(* IEC 61131-3 sources: POMIRTS_lab3/AS/Library_2/AsNxDpM, 3 files *)

(* ---- AsNxDpM.typ ---- *)
TYPE
	nxdpmLifeList_t			: STRUCT			(*life list*)
		node				: ARRAY[0..127] OF USINT;
	END_STRUCT;

	nxdpmDiagData_t			: STRUCT			(*diagnoctic data*)
		status1				: USINT;			(*status1*)
		status2				: USINT;			(*status2*)
		status3				: USINT;			(*status3*)
		address				: USINT;			(*address*)
		identHigh			: USINT;			(*ident high*)
		identLow			: USINT;			(*ident low*)
		blockData			: ARRAY[0..237] OF USINT;
	END_STRUCT;

	nxdpmAddAdrParam_t		: STRUCT			(*additional address parameter*)
		srcType				: USINT;
		srcSize				: USINT;
		destType			: USINT;
		destSize			: USINT;
		addParam			: ARRAY[0..227] OF USINT;
	END_STRUCT;
END_TYPE

(* ---- AsNxDpM.fun ---- *)
{REDUND_CONTEXT} {REDUND_UNREPLICABLE} FUNCTION_BLOCK nxdpmCommand				(*send command*)
	VAR_INPUT
		enable			: BOOL;			(*enables execution*)
		pDevice			: UDINT;		(*interface name given as a pointer, e.g., "SL<x>.SS<y>.IF<z>"*)
		remoteAdr		: UDINT;		(*remote address*)
		syncCommand		: UDINT;		(*sync command*)
		freezeCommand	: UDINT;		(*freeze command*)
		group			: UDINT;		(*group*)
	END_VAR
	VAR
        _state			: UINT;			(*internal variable*)
		_result			: UINT;			(*internal variable*)
        _srcId			: UDINT;		(*internal variable*)
	END_VAR
	VAR_OUTPUT
		status			: UINT;			(*execution status: ERR_OK, ERR_FUB_ENABLE_FALSE, ERR_FUB_BUSY, 0xXXXX = see help*)
		dpStatus		: UDINT;		(*profibus DP stack status*)
	END_VAR
END_FUNCTION_BLOCK

{REDUND_CONTEXT} {REDUND_UNREPLICABLE} FUNCTION_BLOCK nxdpmSetMode				(*set mode*)
	VAR_INPUT
		enable			: BOOL;			(*enables execution*)
		pDevice			: UDINT;		(*interface name given as a pointer, e.g., "SL<x>.SS<y>.IF<z>"*)
		mode			: UDINT;		(*mode to set*)
	END_VAR
	VAR
        _state			: UINT;			(*internal variable*)
		_result			: UINT;			(*internal variable*)
        _srcId			: UDINT;		(*internal variable*)
	END_VAR
	VAR_OUTPUT
		status			: UINT;			(*execution status: ERR_OK, ERR_FUB_ENABLE_FALSE, ERR_FUB_BUSY, 0xXXXX = see help*)
		dpStatus		: UDINT;		(*profibus DP stack status*)
	END_VAR
END_FUNCTION_BLOCK

{REDUND_CONTEXT} {REDUND_UNREPLICABLE} FUNCTION_BLOCK nxdpmActivate			(*activate/deactivate slave*)
	VAR_INPUT
		enable			: BOOL;			(*enables execution*)
		pDevice			: UDINT;		(*interface name given as a pointer, e.g., "SL<x>.SS<y>.IF<z>"*)
		remoteAdr		: UDINT;		(*remote address*)
		activate		: UDINT;		(*activate/deactivate slave*)
	END_VAR
	VAR
        _state			: UINT;			(*internal variable*)
		_result			: UINT;			(*internal variable*)
        _srcId			: UDINT;		(*internal variable*)
	END_VAR
	VAR_OUTPUT
		status			: UINT;			(*execution status: ERR_OK, ERR_FUB_ENABLE_FALSE, ERR_FUB_BUSY, 0xXXXX = see help*)
		dpStatus		: UDINT;		(*profibus DP stack status*)
	END_VAR
END_FUNCTION_BLOCK

{REDUND_CONTEXT} {REDUND_UNREPLICABLE} FUNCTION_BLOCK nxdpmGetDiag				(*get diagnostic*)
	VAR_INPUT
		enable			: BOOL;			(*enables execution*)
		pDevice			: UDINT;		(*interface name given as a pointer, e.g., "SL<x>.SS<y>.IF<z>"*)
		remoteAdr		: UDINT;		(*remote address*)
		flags			: UDINT;		(*flags*)
		pDiagData		: UDINT;		(*diagnostic data given as a pointer*)
	END_VAR
	VAR
        _state			: UINT;			(*internal variable*)
		_result			: UINT;			(*internal variable*)
        _srcId			: UDINT;		(*internal variable*)
	END_VAR
	VAR_OUTPUT
		status			: UINT;			(*execution status: ERR_OK, ERR_FUB_ENABLE_FALSE, ERR_FUB_BUSY, 0xXXXX = see help*)
		dpStatus		: UDINT;		(*profibus DP stack status*)
		diagDataLen		: UDINT;		(*diagnostic data length*)
	END_VAR
END_FUNCTION_BLOCK

{REDUND_CONTEXT} {REDUND_UNREPLICABLE} FUNCTION_BLOCK nxdpmLifeList			(*life list*)
	VAR_INPUT
		enable			: BOOL;			(*enables execution*)
		pDevice			: UDINT;		(*interface name given as a pointer, e.g., "SL<x>.SS<y>.IF<z>"*)
		pLifeList		: UDINT;		(*life list area given as a pointer*)
	END_VAR
	VAR
        _state			: UINT;			(*internal variable*)
		_result			: UINT;			(*internal variable*)
        _srcId			: UDINT;		(*internal variable*)
	END_VAR
	VAR_OUTPUT
		status			: UINT;			(*execution status: ERR_OK, ERR_FUB_ENABLE_FALSE, ERR_FUB_BUSY, 0xXXXX = see help*)
		dpStatus		: UDINT;		(*profibus DP stack status*)
	END_VAR
END_FUNCTION_BLOCK

{REDUND_CONTEXT} {REDUND_UNREPLICABLE} FUNCTION_BLOCK nxdpmV1C1Read			(*DPV1 class 1 read request*)
	VAR_INPUT
		enable			: BOOL;			(*enables execution*)
		pDevice			: UDINT;		(*interface name given as a pointer, e.g., "SL<x>.SS<y>.IF<z>"*)
		remoteAdr		: UDINT;		(*remote address*)
		slotNumber		: UDINT;		(*slot number*)
		index			: UDINT;		(*index*)
		dataLen			: UDINT;		(*data length*)
		pData			: UDINT;		(*data area given as a pointer*)
	END_VAR
	VAR
        _state			: UINT;			(*internal variable*)
		_result			: UINT;			(*internal variable*)
        _srcId			: UDINT;		(*internal variable*)
	END_VAR
	VAR_OUTPUT
		status			: UINT;			(*execution status: ERR_OK, ERR_FUB_ENABLE_FALSE, ERR_FUB_BUSY, 0xXXXX = see help*)
		dpStatus		: UDINT;		(*profibus DP stack status*)
		readDataLen		: UDINT;		(*read data length*)
	END_VAR
END_FUNCTION_BLOCK

{REDUND_CONTEXT} {REDUND_UNREPLICABLE} FUNCTION_BLOCK nxdpmV1C1Write			(*DPV1 class 1 write request*)
	VAR_INPUT
		enable			: BOOL;			(*enables execution*)
		pDevice			: UDINT;		(*interface name given as a pointer, e.g., "SL<x>.SS<y>.IF<z>"*)
		remoteAdr		: UDINT;		(*remote address*)
		slotNumber		: UDINT;		(*slot number*)
		index			: UDINT;		(*index*)
		dataLen			: UDINT;		(*data length*)
		pData			: UDINT;		(*data area given as a pointer*)
	END_VAR
	VAR
        _state			: UINT;			(*internal variable*)
		_result			: UINT;			(*internal variable*)
        _srcId			: UDINT;		(*internal variable*)
	END_VAR
	VAR_OUTPUT
		status			: UINT;			(*execution status: ERR_OK, ERR_FUB_ENABLE_FALSE, ERR_FUB_BUSY, 0xXXXX = see help*)
		dpStatus		: UDINT;		(*profibus DP stack status*)
		errorDecode		: USINT;		(*error decode*)
		errorCode1		: USINT;		(*error code 1*)
		errorCode2		: USINT;		(*error code 2*)
	END_VAR
END_FUNCTION_BLOCK

{REDUND_CONTEXT} {REDUND_UNREPLICABLE} FUNCTION_BLOCK nxdpmSubscribe			(*subscribe master*)
	VAR_INPUT
		enable			: BOOL;			(*enables execution*)
		pDevice			: UDINT;		(*interface name given as a pointer, e.g., "SL<x>.SS<y>.IF<z>"*)
	END_VAR
	VAR
        _state			: UINT;			(*internal variable*)
		_result			: UINT;			(*internal variable*)
        _srcId			: UDINT;		(*internal variable*)
	END_VAR
	VAR_OUTPUT
		status			: UINT;			(*execution status: ERR_OK, ERR_FUB_ENABLE_FALSE, ERR_FUB_BUSY, 0xXXXX = see help*)
		dpStatus		: UDINT;		(*profibus DP stack status*)
	END_VAR
END_FUNCTION_BLOCK

{REDUND_CONTEXT} {REDUND_UNREPLICABLE} FUNCTION_BLOCK nxdpmUnsubscribe			(*unsubscribe master*)
	VAR_INPUT
		enable			: BOOL;			(*enables execution*)
		pDevice			: UDINT;		(*interface name given as a pointer, e.g., "SL<x>.SS<y>.IF<z>"*)
	END_VAR
	VAR
        _state			: UINT;			(*internal variable*)
		_result			: UINT;			(*internal variable*)
        _srcId			: UDINT;		(*internal variable*)
	END_VAR
	VAR_OUTPUT
		status			: UINT;			(*execution status: ERR_OK, ERR_FUB_ENABLE_FALSE, ERR_FUB_BUSY, 0xXXXX = see help*)
		dpStatus		: UDINT;		(*profibus DP stack status*)
	END_VAR
END_FUNCTION_BLOCK

{REDUND_CONTEXT} {REDUND_UNREPLICABLE} FUNCTION_BLOCK nxdpmAlarmReceive		(*receive alarm*)
	VAR_INPUT
		enable			: BOOL;			(*enables execution*)
		pDevice			: UDINT;		(*interface name given as a pointer, e.g., "SL<x>.SS<y>.IF<z>"*)
		remoteAdr		: UDINT;		(*remote address*)
		maxAlarmDataLen	: UDINT;		(*max alarm data length*)
		pAlarmData		: UDINT;		(*alarm data area given as a pointer*)
	END_VAR
	VAR
        _state			: UINT;			(*internal variable*)
		_result			: UINT;			(*internal variable*)
        _srcId			: UDINT;		(*internal variable*)
	END_VAR
	VAR_OUTPUT
		status			: UINT;			(*execution status: ERR_OK, ERR_FUB_ENABLE_FALSE, ERR_FUB_BUSY, 0xXXXX = see help*)
		dpStatus		: UDINT;		(*profibus DP stack status*)
		slotNumber		: USINT;		(*slot number*)
		seqNumber		: USINT;		(*sequence number*)
		alarmType		: USINT;		(*alarm type*)
		alarmSpecifier	: USINT;		(*alarm specifier*)
		addAck			: BOOL;			(*additional acknowledgement flag*)
		alarmDataLen	: UDINT;		(*alarm data length*)
	END_VAR
END_FUNCTION_BLOCK

{REDUND_CONTEXT} {REDUND_UNREPLICABLE} FUNCTION_BLOCK nxdpmAlarmReset			(*reset alarm*)
	VAR_INPUT
		enable			: BOOL;			(*enables execution*)
		pDevice			: UDINT;		(*interface name given as a pointer, e.g., "SL<x>.SS<y>.IF<z>"*)
		remoteAdr		: UDINT;		(*remote address*)
		slotNumber		: USINT;		(*slot number*)
		seqNumber		: USINT;		(*sequence number*)
		alarmType		: USINT;		(*alarm type*)
		alarmSpecifier	: USINT;		(*alarm specifier*)
		addAck			: BOOL;			(*additional acknowledgement flag*)
	END_VAR
	VAR
        _state			: UINT;			(*internal variable*)
		_result			: UINT;			(*internal variable*)
        _srcId			: UDINT;		(*internal variable*)
	END_VAR
	VAR_OUTPUT
		status			: UINT;			(*execution status: ERR_OK, ERR_FUB_ENABLE_FALSE, ERR_FUB_BUSY, 0xXXXX = see help*)
		dpStatus		: UDINT;		(*profibus DP stack status*)
	END_VAR
END_FUNCTION_BLOCK

{REDUND_CONTEXT} {REDUND_UNREPLICABLE} FUNCTION_BLOCK nxdpmV1C2Initiate		(*DPV1 class 2 initiate connection*)
	VAR_INPUT
		enable			: BOOL;			(*enables execution*)
		pDevice			: UDINT;		(*interface name given as a pointer, e.g., "SL<x>.SS<y>.IF<z>"*)
		remoteAdr		: UDINT;		(*remote address*)
		sendTimeout		: UINT;			(*send timeout*)
		featuresSup1	: USINT;		(*service functionality supported*)
		featuresSup2	: USINT;		(*additional service functionality supported*)
		profileFeatSup1	: USINT;		(*profile supported features*)
		profileFeatSup2	: USINT;		(*profile additional supported features*)
		profileIdent	: UINT;			(*profile ident number*)
		pAddAdrParam	: UDINT;		(*additional address parameter given as pointer*)
	END_VAR
	VAR
        _state			: UINT;			(*internal variable*)
		_result			: UINT;			(*internal variable*)
        _srcId			: UDINT;		(*internal variable*)
	END_VAR
	VAR_OUTPUT
		status			: UINT;			(*execution status: ERR_OK, ERR_FUB_ENABLE_FALSE, ERR_FUB_BUSY, 0xXXXX = see help*)
		dpStatus		: UDINT;		(*profibus DP stack status*)
		connectionRef	: UDINT;		(*connection reference*)
		dataUnitSizeMax	: USINT;		(*maximum size of data unit to transfer*)
		slFeaturesSup1	: USINT;		(*service functionality supported by the slave*)
		slFeaturesSup2	: USINT;		(*additional service functionality supported by the slave*)
		slProfFeatSup1	: USINT;		(*supported profile features by the slave*)
		slProfFeatSup2	: USINT;		(*additional supported profile features by the slave*)
		errorDecode		: USINT;
		errorCode1		: USINT;
		errorCode2		: USINT;
		detail			: UINT;
	END_VAR
END_FUNCTION_BLOCK

{REDUND_CONTEXT} {REDUND_UNREPLICABLE} FUNCTION_BLOCK nxdpmV1C2Read			(*DPV1 class 2 read request*)
	VAR_INPUT
		enable			: BOOL;			(*enables execution*)
		pDevice			: UDINT;		(*interface name given as a pointer, e.g., "SL<x>.SS<y>.IF<z>"*)
		connectionRef	: UDINT;		(*connection reference*)
		slotNumber		: UDINT;		(*slot number*)
		index			: UDINT;		(*index*)
		dataLen			: UDINT;		(*number of bytes to read*)
		pData			: UDINT;		(*data area given as a pointer*)
	END_VAR
	VAR
        _state			: UINT;			(*internal variable*)
		_result			: UINT;			(*internal variable*)
        _srcId			: UDINT;		(*internal variable*)
	END_VAR
	VAR_OUTPUT
		status			: UINT;			(*execution status: ERR_OK, ERR_FUB_ENABLE_FALSE, ERR_FUB_BUSY, 0xXXXX = see help*)
		dpStatus		: UDINT;		(*profibus DP stack status*)
		readDataLen		: UDINT;		(*read data length*)
		errorDecode		: USINT;
		errorCode1		: USINT;
		errorCode2		: USINT;
	END_VAR
END_FUNCTION_BLOCK

{REDUND_CONTEXT} {REDUND_UNREPLICABLE} FUNCTION_BLOCK nxdpmV1C2Write			(*DPV1 class 2 write request*)
	VAR_INPUT
		enable			: BOOL;			(*enables execution*)
		pDevice			: UDINT;		(*interface name given as a pointer, e.g., "SL<x>.SS<y>.IF<z>"*)
		connectionRef	: UDINT;		(*connection reference*)
		slotNumber		: UDINT;		(*slot number*)
		index			: UDINT;		(*index*)
		dataLen			: UDINT;		(*number of bytes to write*)
		pData			: UDINT;		(*data area given as a pointer*)
	END_VAR
	VAR
        _state			: UINT;			(*internal variable*)
		_result			: UINT;			(*internal variable*)
        _srcId			: UDINT;		(*internal variable*)
	END_VAR
	VAR_OUTPUT
		status			: UINT;			(*execution status: ERR_OK, ERR_FUB_ENABLE_FALSE, ERR_FUB_BUSY, 0xXXXX = see help*)
		dpStatus		: UDINT;		(*profibus DP stack status*)
		errorDecode		: USINT;
		errorCode1		: USINT;
		errorCode2		: USINT;
	END_VAR
END_FUNCTION_BLOCK

{REDUND_CONTEXT} {REDUND_UNREPLICABLE} FUNCTION_BLOCK nxdpmV1C2Data			(*combined DPV1 class 2 read and write request*)
	VAR_INPUT
		enable			: BOOL;			(*enables execution*)
		pDevice			: UDINT;		(*interface name given as a pointer, e.g., "SL<x>.SS<y>.IF<z>"*)
		connectionRef	: UDINT;		(*connection reference*)
		slotNumber		: UDINT;		(*slot number*)
		index			: UDINT;		(*index*)
		dataLen			: UDINT;		(*number of bytes to write*)
		pDataWrite		: UDINT;		(*write data area given as a pointer*)
		pDataRead		: UDINT;		(*read data area given as a pointer*)
	END_VAR
	VAR
        _state			: UINT;			(*internal variable*)
		_result			: UINT;			(*internal variable*)
        _srcId			: UDINT;		(*internal variable*)
	END_VAR
	VAR_OUTPUT
		status			: UINT;			(*execution status: ERR_OK, ERR_FUB_ENABLE_FALSE, ERR_FUB_BUSY, 0xXXXX = see help*)
		dpStatus		: UDINT;		(*profibus DP stack status*)
		readDataLen		: UDINT;		(*read data length*)
		errorDecode		: USINT;
		errorCode1		: USINT;
		errorCode2		: USINT;
	END_VAR
END_FUNCTION_BLOCK

{REDUND_CONTEXT} {REDUND_UNREPLICABLE} FUNCTION_BLOCK nxdpmV1C2Abort			(*V1 class 2 request abort of connection*)
	VAR_INPUT
		enable			: BOOL;			(*enables execution*)
		pDevice			: UDINT;		(*interface name given as a pointer, e.g., "SL<x>.SS<y>.IF<z>"*)
		connectionRef	: UDINT;		(*connection reference*)
		subnet			: USINT;		(*subnet*)
		instance		: USINT;		(*instance number*)
		reasonCode		: USINT;		(*reason code why an abort is requested*)
	END_VAR
	VAR
        _state			: UINT;			(*internal variable*)
		_result			: UINT;			(*internal variable*)
        _srcId			: UDINT;		(*internal variable*)
	END_VAR
	VAR_OUTPUT
		status			: UINT;			(*execution status: ERR_OK, ERR_FUB_ENABLE_FALSE, ERR_FUB_BUSY, 0xXXXX = see help*)
		dpStatus		: UDINT;		(*profibus DP stack status*)
	END_VAR
END_FUNCTION_BLOCK

(* ---- AsNxDpM.var ---- *)
VAR CONSTANT
	nxdpmERR_INVALID_DEVICE					: UINT	:= 34700;		(*error invalid device*)
	nxdpmERR_SEND_MESSAGE					: UINT	:= 34701;		(*error send message*)
	nxdpmERR_TIMEOUT						: UINT	:= 34702;		(*error timeout*)
	nxdpmERR_PROFIBUSDP_STACK				: UINT	:= 34703;		(*error receive message*)
	nxdpmERR_PARAMETER						: UINT	:= 34704;		(*error invalid parameter*)
	nxdpmERR_MEMORY							: UINT	:= 34705;		(*error less memory*)
	nxdpmERR_SUBSCRIBE_LISTENER				: UINT	:= 34706;		(*error subscribe listener*)
	nxdpmERR_NO_MORE_ENTRIES				: UINT	:= 34707;		(*error no more entries available*)

	nxdpmCMD_UNFREEZE						: UDINT	:= 4;			(*unfreeze command*)
	nxdpmCMD_FREEZE							: UDINT	:= 8;			(*freeze command*)
	nxdpmCMD_UNSYNC							: UDINT	:= 16;			(*unsync command*)
	nxdpmCMD_SYNC							: UDINT	:= 32;			(*sync command*)

	nxdpmMODE_OFFLINE						: UDINT	:= 16#00000000;	(*mode offline*)
	nxdpmMODE_STOP							: UDINT	:= 16#00000040;	(*mode stop*)
	nxdpmMODE_CLEAR							: UDINT	:= 16#00000080;	(*mode clear*)
	nxdpmMODE_OPERATE						: UDINT	:= 16#000000C0;	(*mode operate*)

	nxdpmFLAG_PEEK							: UDINT	:= 16#00000001;	(*node remains in diagnostic lists after request*)
	nxdpmFLAG_QUERY							: UDINT	:= 16#00000002;	(*get diagnostic direct from slave*)

	nxdpmFLAG_STATION_NON_EXISTENT			: USINT	:= 16#01;		(*station non existent*)
	nxdpmFLAG_STATION_NOT_READY				: USINT	:= 16#02;		(*station not ready*)
	nxdpmFLAG_CFG_FAULT						: USINT	:= 16#04;		(*configuration fault*)
	nxdpmFLAG_EXT_DIAG						: USINT	:= 16#08;		(*extended diagnostic*)
	nxdpmFLAG_NOT_SUPPORTED					: USINT	:= 16#10;		(*not supported*)
	nxdpmFLAG_INVALID_SLAVE_RESPONSE		: USINT	:= 16#20;		(*invalid slave response*)
	nxdpmFLAG_PRM_FAULT						: USINT	:= 16#40;		(*parameter fault*)
	nxdpmFLAG_MASTER_LOCK					: USINT	:= 16#80;		(*master lock*)

	nxdpmFLAG_PRM_REQUEST					: USINT	:= 16#01;		(*parameter request*)
	nxdpmFLAG_STAT_DIAG						: USINT	:= 16#02;		(*statistical diagnosis*)
	nxdpmFLAG_1								: USINT	:= 16#04;		(*this bit is always set to the value 1 indicating DP V1 operation*)
	nxdpmFLAG_WD_ON							: USINT	:= 16#08;		(*watchdog activated*)
	nxdpmFLAG_FREEZE_MODE					: USINT	:= 16#10;		(*freeze mode*)
	nxdpmFLAG_SYNC_MODE						: USINT	:= 16#20;		(*sync mode*)
	nxdpmFLAG_DEACTIVATED					: USINT	:= 16#80;		(*non projected slave*)

	nxdpmFLAG_EXT_DIAG_OVERFLOW				: USINT	:= 16#80;		(*this bit indicates that the slave has more diagnostic data available than it can send*)

	nxdpmLIFE_LIST_SIZE						: UDINT	:= 128;			(*size of life list*)
	nxdpmNODE_NOT_PRESENT					: UDINT	:= 0;			(*not present*)
	nxdpmNODE_SLAVE							: UDINT	:= 1;			(*slave*)
	nxdpmNODE_MASTER						: UDINT	:= 3;			(*master*)

	nxdpmACTIVATE							: UDINT	:= 1;			(*activate slave*)
	nxdpmDEACTIVATE							: UDINT	:= 2;			(*deactivate slave*)

	nxdpmALARM_DIAGNOSTIC					: USINT	:= 1;			(*diagnostic alarm*)
	nxdpmALARM_PROCESS						: USINT	:= 2;			(*process alarm*)
	nxdpmALARM_PULL							: USINT	:= 3;			(*pull alarm*)
	nxdpmALARM_PLUG							: USINT	:= 4;			(*plug alarm*)
	nxdpmALARM_STATUS						: USINT	:= 5;			(*status alarm*)
	nxdpmALARM_UPDATE						: USINT	:= 6;			(*update alarm*)

	nxdpmALARM_SPEC_NO_DIFF					: USINT	:= 0;			(*no further differentiation*)
	nxdpmALARM_SPEC_ERR_APP_SLOT_DIS		: USINT	:= 1;			(*error appears and slot disturbed*)
	nxdpmALARM_SPEC_ERR_DIS_SLOT_OK			: USINT	:= 2;			(*error disappears and slot is ok*)
	nxdpmALARM_SPEC_ERR_DIS_SLOT_DIS		: USINT	:= 3;			(*error disappears and slot is still disturbed*)
END_VAR
